FUNCTION_BLOCK RT_E_DELAY (* Delayed propagation of an event-Cancellable *)
  (* Description: Copyright (c) 2008, 2014 ACIN, Profactor GmbH This program and the accompanying materials are made available under the terms of the Eclipse Public License 2.0 which is available at https://www.eclipse.org/legal/epl-2.0/ SPDX-License-Identifier: EPL-2.0 *)
  (* Version 1.0, 2008-07-10, Alois Zoitl, ACIN *)
  (* Version 1.1, 2011-06-04, Alois Zoitl, Profactor GmbH *)
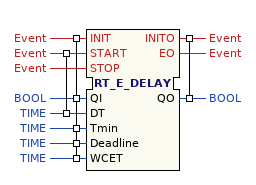
  EVENT_INPUT
    INIT WITH QI, Tmin, Deadline, WCET;
    START WITH DT; (* Begin Delay *)
    STOP; (* Cancel Delay *)
  END_EVENT
  EVENT_OUTPUT
    INITO WITH QO;
    EO; (* Delayed Event *)
  END_EVENT
  VAR_INPUT
    QI : BOOL;
    DT : TIME; (* Delay Time *)
    Tmin : TIME;
    Deadline : TIME;
    WCET : TIME;
  END_VAR
  VAR_OUTPUT
    QO : BOOL;
  END_VAR
END_FUNCTION_BLOCK
